// TIA Portal V17 export
// export: Created 2025-06-25T13:13:12.9539777Z, ExportSetting WithDefaults, DisplayName Totally Integrated Automation Portal, DisplayVersion V17 Update 8, DisplayName TIA Portal Openness, DisplayVersion V17 Update 8, DisplayName TIA Portal Version Control Interface, DisplayVersion V17, DisplayName STEP 7 Professional, DisplayVersion V17 Update 8, DisplayName STEP 7 Safety, DisplayVersion V17 Update 6, DisplayName WinCC Advanced, DisplayVersion V17 Update 8
FUNCTION_BLOCK "Diagnosis"   // FB1, FBD
TITLE = Misc alarm handling
{ S7_Optimized_Access := 'TRUE' }
VERSION : 0.1
// stored: AutoNumber true, IsIECCheckEnabled false, IsRetainMemResEnabled false, MemoryReserve 0, SetENOAutomatically false, UDAEnableTagReadback false
   VAR
      A0001 { ExternalAccessible := 'False'; ExternalVisible := 'False'; ExternalWritable := 'False'} : "fbHMIEvent";
      A1002 { ExternalAccessible := 'False'; ExternalVisible := 'False'; ExternalWritable := 'False'; S7_SetPoint := 'True'} : "fbHMIEvent";
      A1003 { ExternalAccessible := 'False'; ExternalVisible := 'False'; ExternalWritable := 'False'; S7_SetPoint := 'True'} : "fbHMIEvent";
   END_VAR
BEGIN

REGION Network 1: 0001 Watchdog timeout OB1
   // "DB_Alarms"."0001_WatchdogTimeoutOB1".bInput is written by OB80, but alarm is processed here (OB80 is not cyclic)
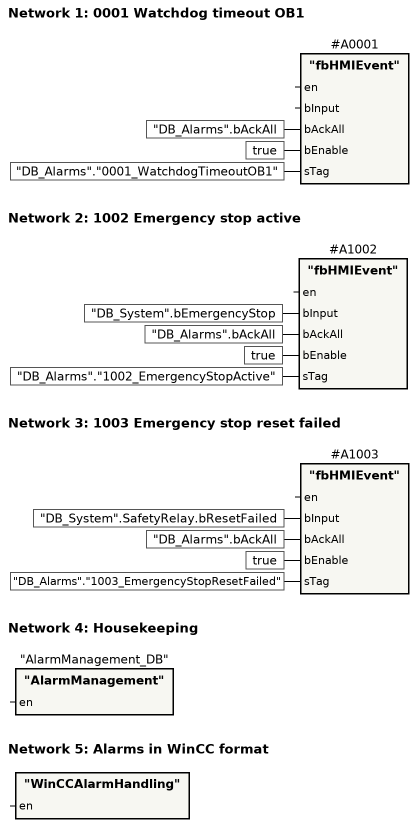
   #A0001(bAckAll := "DB_Alarms".bAckAll, bEnable := true, sTag := "DB_Alarms"."0001_WatchdogTimeoutOB1");   // "fbHMIEvent"
END_REGION

REGION Network 2: 1002 Emergency stop active
   #A1002(bInput := "DB_System".bEmergencyStop,   // "fbHMIEvent"
          bAckAll := "DB_Alarms".bAckAll,
          bEnable := true,
          sTag := "DB_Alarms"."1002_EmergencyStopActive");
END_REGION

REGION Network 3: 1003 Emergency stop reset failed
   #A1003(bInput := "DB_System".SafetyRelay.bResetFailed,   // "fbHMIEvent"
          bAckAll := "DB_Alarms".bAckAll,
          bEnable := true,
          sTag := "DB_Alarms"."1003_EmergencyStopResetFailed");
END_REGION

REGION Network 4: Housekeeping
   "AlarmManagement_DB"();   // "AlarmManagement"
END_REGION

REGION Network 5: Alarms in WinCC format
   "WinCCAlarmHandling"();
END_REGION

REGION Network 6 (SCL): Alarms to App PLC - Group 0 & 1
   // Group 0-System
   "DB_Application".FromHB.Alarms[0] := "DB_WinCCAlarms"."0-System"."0001_WatchdogTimeoutOB1".Memory.%X0;
   "DB_Application".FromHB.Alarms[1] := "DB_WinCCAlarms"."0-System"."0003_InitCurrenSettingsFailed".Memory.%X0;
   "DB_Application".FromHB.Alarms[2] := "DB_WinCCAlarms"."0-System"."0006_CPUinErrorState".Memory.%X0;

   // Group 1-IO
   "DB_Application".FromHB.Alarms[3]  := "DB_WinCCAlarms"."1-IO"."1001_ConnectionToWinCClost".Memory.%X0;
   "DB_Application".FromHB.Alarms[4]  := "DB_WinCCAlarms"."1-IO"."1002_EmergencyStopActive".Memory.%X0;
   "DB_Application".FromHB.Alarms[5]  := "DB_WinCCAlarms"."1-IO"."1003_SafetyRelayResetFailed".Memory.%X0;
   "DB_Application".FromHB.Alarms[6]  := "DB_WinCCAlarms"."1-IO"."1004_HBL_PS_01_X2".Memory.%X0;
   "DB_Application".FromHB.Alarms[7]  := "DB_WinCCAlarms"."1-IO"."1101_HBL_SC_01_CommError".Memory.%X0;
   "DB_Application".FromHB.Alarms[8]  := "DB_WinCCAlarms"."1-IO"."1102_HBL_SC_02_CommError".Memory.%X0;
   "DB_Application".FromHB.Alarms[9]  := "DB_WinCCAlarms"."1-IO"."1110_HBL_SC_10_CommError".Memory.%X0;
   "DB_Application".FromHB.Alarms[10] := "DB_WinCCAlarms"."1-IO"."1121_HBL_SC_01_Tripped".Memory.%X0;
   "DB_Application".FromHB.Alarms[11] := "DB_WinCCAlarms"."1-IO"."1122_HBL_SC_02_Tripped".Memory.%X0;
   "DB_Application".FromHB.Alarms[12] := "DB_WinCCAlarms"."1-IO"."1130_HBL_SC_10_Tripped".Memory.%X0;
   "DB_Application".FromHB.Alarms[13] := "DB_WinCCAlarms"."1-IO"."1140_HBL_SC_01_RunFailure".Memory.%X0;
   "DB_Application".FromHB.Alarms[14] := "DB_WinCCAlarms"."1-IO"."1142_HBL_SC_02_RunFailure".Memory.%X0;
   "DB_Application".FromHB.Alarms[15] := "DB_WinCCAlarms"."1-IO"."1150_HBL_SC_10_RunFailure".Memory.%X0;

   "DB_Application".FromHB.Alarms[16] := "DB_WinCCAlarms"."1-IO"."1201_HBL_PT_01_Fault".Memory.%X0;
   "DB_Application".FromHB.Alarms[17] := "DB_WinCCAlarms"."1-IO"."1202_HBL_PT_02_Fault".Memory.%X0;
   "DB_Application".FromHB.Alarms[18] := "DB_WinCCAlarms"."1-IO"."1203_HBL_PT_03_Fault".Memory.%X0;
   "DB_Application".FromHB.Alarms[19] := "DB_WinCCAlarms"."1-IO"."1204_HBL_PT_04_Fault".Memory.%X0;
   "DB_Application".FromHB.Alarms[20] := "DB_WinCCAlarms"."1-IO"."1205_HBL_TT_05_Fault".Memory.%X0;
   "DB_Application".FromHB.Alarms[21] := "DB_WinCCAlarms"."1-IO"."1206_HBL_TT_06_Fault".Memory.%X0;
   "DB_Application".FromHB.Alarms[22] := "DB_WinCCAlarms"."1-IO"."1207_HBL_TT_07_Fault".Memory.%X0;
   "DB_Application".FromHB.Alarms[23] := "DB_WinCCAlarms"."1-IO"."1208_HBL_TT_08_Fault".Memory.%X0;
   "DB_Application".FromHB.Alarms[24] := "DB_WinCCAlarms"."1-IO"."1209_HBL_HCV_01_A1_Fault".Memory.%X0;
   "DB_Application".FromHB.Alarms[25] := "DB_WinCCAlarms"."1-IO"."1210_HBL_TT_10_Fault".Memory.%X0;
   "DB_Application".FromHB.Alarms[26] := "DB_WinCCAlarms"."1-IO"."1212_HBL_TT_12_Fault".Memory.%X0;
   "DB_Application".FromHB.Alarms[27] := "DB_WinCCAlarms"."1-IO"."1213_HBL_TT_13_Fault".Memory.%X0;
   "DB_Application".FromHB.Alarms[28] := "DB_WinCCAlarms"."1-IO"."1214_HBL_TT_14_Fault".Memory.%X0;
   "DB_Application".FromHB.Alarms[29] := "DB_WinCCAlarms"."1-IO"."1215_HBL_TT_15_Fault".Memory.%X0;
   "DB_Application".FromHB.Alarms[30] := "DB_WinCCAlarms"."1-IO"."1216_HBL_TT_16_Fault".Memory.%X0;
   "DB_Application".FromHB.Alarms[31] := "DB_WinCCAlarms"."1-IO"."1217_HBL_TT_17_Fault".Memory.%X0;
   "DB_Application".FromHB.Alarms[32] := "DB_WinCCAlarms"."1-IO"."1218_HBL_TT_18_Fault".Memory.%X0;
   "DB_Application".FromHB.Alarms[33] := "DB_WinCCAlarms"."1-IO"."1220_HBL_PT_960_Fault".Memory.%X0;
   "DB_Application".FromHB.Alarms[34] := "DB_WinCCAlarms"."1-IO"."1221_HBL_PT_05_Fault".Memory.%X0;
   "DB_Application".FromHB.Alarms[35] := "DB_WinCCAlarms"."1-IO"."1223_HBL_TT_03_Fault".Memory.%X0;
   "DB_Application".FromHB.Alarms[36] := "DB_WinCCAlarms"."1-IO"."1224_HBL_TT_23_Fault".Memory.%X0;
   "DB_Application".FromHB.Alarms[37] := "DB_WinCCAlarms"."1-IO"."1225_HBL_TT_24_Fault".Memory.%X0;
   "DB_Application".FromHB.Alarms[38] := "DB_WinCCAlarms"."1-IO"."1226_HBL_TT_25_Fault".Memory.%X0;
   "DB_Application".FromHB.Alarms[39] := "DB_WinCCAlarms"."1-IO"."1227_HBL_LT_01_Fault".Memory.%X0;
   "DB_Application".FromHB.Alarms[40] := "DB_WinCCAlarms"."1-IO"."1228_HBL_TT_21_Fault".Memory.%X0;
   "DB_Application".FromHB.Alarms[41] := "DB_WinCCAlarms"."1-IO"."1229_HBL_TT_22_Fault".Memory.%X0;
   "DB_Application".FromHB.Alarms[42] := "DB_WinCCAlarms"."1-IO"."1230_HBL_LT_02_Fault".Memory.%X0;
   "DB_Application".FromHB.Alarms[43] := "DB_WinCCAlarms"."1-IO"."1231_HBL_HCV_02_A1_Fault".Memory.%X0;
   "DB_Application".FromHB.Alarms[44] := "DB_WinCCAlarms"."1-IO"."1232_HBL_PT_13_Fault".Memory.%X0;
   "DB_Application".FromHB.Alarms[45] := "DB_WinCCAlarms"."1-IO"."1233_HBL_TT_20_Fault".Memory.%X0;
   "DB_Application".FromHB.Alarms[46] := "DB_WinCCAlarms"."1-IO"."1234_HBL_PT_14_Fault".Memory.%X0;
   "DB_Application".FromHB.Alarms[47] := "DB_WinCCAlarms"."1-IO"."1235_HBL_PT_18_Fault".Memory.%X0;
   "DB_Application".FromHB.Alarms[48] := "DB_WinCCAlarms"."1-IO"."1236_HBL_PT_19_Fault".Memory.%X0;
   "DB_Application".FromHB.Alarms[49] := "DB_WinCCAlarms"."1-IO"."1237_HBL_PT_25_Fault".Memory.%X0;
   "DB_Application".FromHB.Alarms[50] := "DB_WinCCAlarms"."1-IO"."1238_HBL_TT_31_Fault".Memory.%X0;
   "DB_Application".FromHB.Alarms[51] := "DB_WinCCAlarms"."1-IO"."1239_HBL_TT_33_Fault".Memory.%X0;
   "DB_Application".FromHB.Alarms[52] := "DB_WinCCAlarms"."1-IO"."1240_HBL_TT_35_Fault".Memory.%X0;
   "DB_Application".FromHB.Alarms[53] := "DB_WinCCAlarms"."1-IO"."1241_HBL_HCV_01_Fault".Memory.%X0;
   "DB_Application".FromHB.Alarms[54] := "DB_WinCCAlarms"."1-IO"."1242_HBL_HCV_02_Fault".Memory.%X0;
   "DB_Application".FromHB.Alarms[55] := "DB_WinCCAlarms"."1-IO"."1243_HBL_PT_07_Fault".Memory.%X0;
   "DB_Application".FromHB.Alarms[56] := "DB_WinCCAlarms"."1-IO"."1244_HBL_PT_08_Fault".Memory.%X0;
   "DB_Application".FromHB.Alarms[57] := "DB_WinCCAlarms"."1-IO"."1245_HBL_PT_09_Fault".Memory.%X0;
   "DB_Application".FromHB.Alarms[58] := "DB_WinCCAlarms"."1-IO"."1246_HBL_PT_10_Fault".Memory.%X0;
   "DB_Application".FromHB.Alarms[59] := "DB_WinCCAlarms"."1-IO"."1247_HBL_PT_11_Fault".Memory.%X0;
   "DB_Application".FromHB.Alarms[60] := "DB_WinCCAlarms"."1-IO"."1248_HBL_PT_12_Fault".Memory.%X0;
   "DB_Application".FromHB.Alarms[61] := "DB_WinCCAlarms"."1-IO"."1249_HBL_PT_15_Fault".Memory.%X0;
   "DB_Application".FromHB.Alarms[62] := FALSE;
   "DB_Application".FromHB.Alarms[63] := "DB_WinCCAlarms"."1-IO"."1251_HBL_PT_24_Fault".Memory.%X0;
   "DB_Application".FromHB.Alarms[64] := "DB_WinCCAlarms"."1-IO"."1252_HBL_TT_28_Fault".Memory.%X0;
   "DB_Application".FromHB.Alarms[65] := "DB_WinCCAlarms"."1-IO"."1253_HBL_TT_29_Fault".Memory.%X0;
   "DB_Application".FromHB.Alarms[66] := "DB_WinCCAlarms"."1-IO"."1254_HBL_TT_32_Fault".Memory.%X0;
   "DB_Application".FromHB.Alarms[67] := "DB_WinCCAlarms"."1-IO"."1255_HBL_CT_01_Fault".Memory.%X0;
   "DB_Application".FromHB.Alarms[68] := "DB_WinCCAlarms"."1-IO"."1256_HBL_CT_02_Fault".Memory.%X0;
   "DB_Application".FromHB.Alarms[69] := FALSE;
   "DB_Application".FromHB.Alarms[70] := "DB_WinCCAlarms"."1-IO"."1258_HBL_TT_26_Fault".Memory.%X0;
   "DB_Application".FromHB.Alarms[71] := "DB_WinCCAlarms"."1-IO"."1259_HBL_TT_27_Fault".Memory.%X0;
   "DB_Application".FromHB.Alarms[72] := "DB_WinCCAlarms"."1-IO"."1260_HBL_FT_01_Fault".Memory.%X0;
   "DB_Application".FromHB.Alarms[73] := FALSE;
   "DB_Application".FromHB.Alarms[74] := "DB_WinCCAlarms"."1-IO"."1262_HBL_TT_30_Fault".Memory.%X0;
   "DB_Application".FromHB.Alarms[75] := "DB_WinCCAlarms"."1-IO"."1263_HBL_TT_34_Fault".Memory.%X0;
   "DB_Application".FromHB.Alarms[76] := "DB_WinCCAlarms"."1-IO"."1264".Memory.%X0;
END_REGION

REGION Network 7 (SCL): Alarms to App PLC - Group 2
   "DB_Application".FromHB.Alarms[77] := "DB_WinCCAlarms"."2-ProcessValues"."2018".Memory.%X0;
   "DB_Application".FromHB.Alarms[78] := "DB_WinCCAlarms"."2-ProcessValues"."2028".Memory.%X0;
   "DB_Application".FromHB.Alarms[79] := "DB_WinCCAlarms"."2-ProcessValues"."2058".Memory.%X0;
   "DB_Application".FromHB.Alarms[80] := "DB_WinCCAlarms"."2-ProcessValues"."2100".Memory.%X0;
   "DB_Application".FromHB.Alarms[81] := "DB_WinCCAlarms"."2-ProcessValues"."2101".Memory.%X0;
   "DB_Application".FromHB.Alarms[82] := "DB_WinCCAlarms"."2-ProcessValues"."2102".Memory.%X0;
   "DB_Application".FromHB.Alarms[83] := "DB_WinCCAlarms"."2-ProcessValues"."2103".Memory.%X0;
   "DB_Application".FromHB.Alarms[84] := "DB_WinCCAlarms"."2-ProcessValues"."2105".Memory.%X0;
   "DB_Application".FromHB.Alarms[85] := "DB_WinCCAlarms"."2-ProcessValues"."2106".Memory.%X0;
   "DB_Application".FromHB.Alarms[86] := "DB_WinCCAlarms"."2-ProcessValues"."2107".Memory.%X0;
   "DB_Application".FromHB.Alarms[87] := "DB_WinCCAlarms"."2-ProcessValues"."2108".Memory.%X0;
   "DB_Application".FromHB.Alarms[88] := "DB_WinCCAlarms"."2-ProcessValues"."2109".Memory.%X0;
   "DB_Application".FromHB.Alarms[89] := "DB_WinCCAlarms"."2-ProcessValues"."2110".Memory.%X0;
   "DB_Application".FromHB.Alarms[90] := "DB_WinCCAlarms"."2-ProcessValues"."2111".Memory.%X0;
   "DB_Application".FromHB.Alarms[91] := "DB_WinCCAlarms"."2-ProcessValues"."2112".Memory.%X0;
   "DB_Application".FromHB.Alarms[92] := "DB_WinCCAlarms"."2-ProcessValues"."2113".Memory.%X0;
   "DB_Application".FromHB.Alarms[93] := "DB_WinCCAlarms"."2-ProcessValues"."2114".Memory.%X0;
   "DB_Application".FromHB.Alarms[94] := "DB_WinCCAlarms"."2-ProcessValues"."2115".Memory.%X0;
   "DB_Application".FromHB.Alarms[95] := "DB_WinCCAlarms"."2-ProcessValues"."2116".Memory.%X0;
   "DB_Application".FromHB.Alarms[96] := "DB_WinCCAlarms"."2-ProcessValues"."2117".Memory.%X0;
   "DB_Application".FromHB.Alarms[97] := "DB_WinCCAlarms"."2-ProcessValues"."2301_HeatSourceTempDropCritical".Memory.%X0;
   "DB_Application".FromHB.Alarms[98] := "DB_WinCCAlarms"."2-ProcessValues"."2302_HeatSourceTempRiseCritical".Memory.%X0;
   "DB_Application".FromHB.Alarms[99] := "DB_WinCCAlarms"."2-ProcessValues"."2303_SuperheatCompressorHigh".Memory.%X0;
   "DB_Application".FromHB.Alarms[100] := "DB_WinCCAlarms"."2-ProcessValues"."2304_SuperheatCompressorLow".Memory.%X0;
   "DB_Application".FromHB.Alarms[101] := "DB_WinCCAlarms"."2-ProcessValues"."2305_OilFilterDeltaPHigh".Memory.%X0;
   "DB_Application".FromHB.Alarms[102] := "DB_WinCCAlarms"."2-ProcessValues"."2306_OilFilterDeltaPHighHigh".Memory.%X0;
   "DB_Application".FromHB.Alarms[103] := "DB_WinCCAlarms"."2-ProcessValues"."2307_EvaporatorDischargePressureMeanValue".Memory.%X0;
   "DB_Application".FromHB.Alarms[104] := "DB_WinCCAlarms"."2-ProcessValues"."2308_EvaporatorDischargePressureHigh".Memory.%X0;
END_REGION

REGION Network 8 (SCL): Alarms to App PLC - Group 3 & 5
   // Group 3-Control
   "DB_Application".FromHB.Alarms[105] := FALSE; // 3000
   "DB_Application".FromHB.Alarms[106] := "DB_WinCCAlarms"."3-Control"."3020".Memory.%X0;
   "DB_Application".FromHB.Alarms[107] := FALSE; // 3030
   "DB_Application".FromHB.Alarms[108] := FALSE; // 3040
   "DB_Application".FromHB.Alarms[109] := FALSE; // 3050
   "DB_Application".FromHB.Alarms[110] := FALSE; // 3060
   "DB_Application".FromHB.Alarms[111] := FALSE; // 3070
   "DB_Application".FromHB.Alarms[112] := FALSE; // 3080
   "DB_Application".FromHB.Alarms[113] := FALSE; // 3090
   "DB_Application".FromHB.Alarms[114] := FALSE; // 3100
   "DB_Application".FromHB.Alarms[115] := FALSE; // 3110
   "DB_Application".FromHB.Alarms[116] := "DB_WinCCAlarms"."3-Control"."3400_HydrolockProtectionActive".Memory.%X0;
   "DB_Application".FromHB.Alarms[158] := "DB_WinCCAlarms"."3-Control"."3401_DripPanLevelHigh".Memory.%X0;

   // Group 5-Auxiliaries
   "DB_Application".FromHB.Alarms[117] := "DB_WinCCAlarms"."5-Auxiliaries"."5000_OilHeatingActivationFailure".Memory.%X0;
   "DB_Application".FromHB.Alarms[118] := "DB_WinCCAlarms"."5-Auxiliaries"."5001_OilHeatingDeactivationFailure".Memory.%X0;
   "DB_Application".FromHB.Alarms[119] := "DB_WinCCAlarms"."5-Auxiliaries"."5200".Memory.%X0;
   "DB_Application".FromHB.Alarms[120] := "DB_WinCCAlarms"."5-Auxiliaries"."5201".Memory.%X0;
   "DB_Application".FromHB.Alarms[121] := "DB_WinCCAlarms"."5-Auxiliaries"."5202".Memory.%X0;
   "DB_Application".FromHB.Alarms[122] := "DB_WinCCAlarms"."5-Auxiliaries"."5203_CPC_SC_01_CommError".Memory.%X0;
   "DB_Application".FromHB.Alarms[123] := "DB_WinCCAlarms"."5-Auxiliaries"."5204_CPC_SC_01_Tripped".Memory.%X0;
   "DB_Application".FromHB.Alarms[124] := "DB_WinCCAlarms"."5-Auxiliaries"."5205".Memory.%X0;
   "DB_Application".FromHB.Alarms[125] := "DB_WinCCAlarms"."5-Auxiliaries"."5206".Memory.%X0;
   "DB_Application".FromHB.Alarms[126] := "DB_WinCCAlarms"."5-Auxiliaries"."5250_SSC_TT_01_Fault".Memory.%X0;
   "DB_Application".FromHB.Alarms[127] := "DB_WinCCAlarms"."5-Auxiliaries"."5251_SSC_TT_02_Fault".Memory.%X0;
   "DB_Application".FromHB.Alarms[128] := "DB_WinCCAlarms"."5-Auxiliaries"."5252_SSC_TT_03_Fault".Memory.%X0;
   "DB_Application".FromHB.Alarms[129] := "DB_WinCCAlarms"."5-Auxiliaries"."5253_SSC_TT_04_Fault".Memory.%X0;
   "DB_Application".FromHB.Alarms[130] := "DB_WinCCAlarms"."5-Auxiliaries"."5254_SSC_PIT_01_Fault".Memory.%X0;
   "DB_Application".FromHB.Alarms[131] := "DB_WinCCAlarms"."5-Auxiliaries"."5255_SSC_PDT_01_Fault".Memory.%X0;
   "DB_Application".FromHB.Alarms[132] := "DB_WinCCAlarms"."5-Auxiliaries"."5256_SSC_LT_01_Fault".Memory.%X0;
   "DB_Application".FromHB.Alarms[133] := "DB_WinCCAlarms"."5-Auxiliaries"."5257_SSC_LT_01_Low".Memory.%X0;
   "DB_Application".FromHB.Alarms[134] := "DB_WinCCAlarms"."5-Auxiliaries"."5258_SSC_PDT_01_High".Memory.%X0;
   "DB_Application".FromHB.Alarms[135] := "DB_WinCCAlarms"."5-Auxiliaries"."5259_SSC_TT_02_High".Memory.%X0;
   "DB_Application".FromHB.Alarms[136] := "DB_WinCCAlarms"."5-Auxiliaries"."5260_SSC_TT_03_Low".Memory.%X0;
   "DB_Application".FromHB.Alarms[137] := "DB_WinCCAlarms"."5-Auxiliaries"."5261_SSC_PIT_01_Low".Memory.%X0;
   "DB_Application".FromHB.Alarms[138] := "DB_WinCCAlarms"."5-Auxiliaries"."5262_DeltaT_ShaftSealHigh".Memory.%X0;
   "DB_Application".FromHB.Alarms[139] := "DB_WinCCAlarms"."5-Auxiliaries"."5263_SSC_PIT_01_High".Memory.%X0;
   "DB_Application".FromHB.Alarms[140] := "DB_WinCCAlarms"."5-Auxiliaries"."5268_ShaftSealSystemShutdown".Memory.%X0;
END_REGION

REGION Network 9 (SCL): Alarms to App PLC - Group 8
   // Group 8-Events
   //"DB_Application".Status.Alarms[141] := "DB_WinCCAlarms"."8-Events"."8000_State0_Initialize".Memory.%X0;
   //"DB_Application".Status.Alarms[142] := "DB_WinCCAlarms"."8-Events"."8001_State1_Offline".Memory.%X0;
   "DB_Application".FromHB.Alarms[143] := "DB_WinCCAlarms"."8-Events"."8002_State2_Standby".Memory.%X0;
END_REGION
END_FUNCTION_BLOCK
